INTERFACE IPLCOpenGroup

METHOD AbortPreviousCommands : BOOL
VAR_INPUT
	newCommand : IPLCOpenCommand;
END_VAR
END_METHOD

END_INTERFACE

(* stored: Version 1.1.0.1, ProductVersion 3.1.4024.12
   Itf IPLCOpenGroup: Id {b35eb493-5dd7-45b9-9e67-a673072a60b4}
   Method AbortPreviousCommands: Id {33d62d2b-227e-4998-b717-c18b2f1e35eb} *)
